Staubli VAL3: CopyFileContext.pgx

public program CopyFileContext(bool x_bRes (dimensions=1), string x_sFileSource (dimensions=1), string x_sFileDest (dimensions=1), num x_nStart (dimensions=1), num x_nEnd (dimensions=1))
  local num l_nIndex
  local num l_nNum
  local string l_sBuff
begin

  x_bRes=false
  if x_nEnd==-1
    x_nEnd=50000000
  endIf
  if x_sFileDest=="" or x_nStart<0 or x_nEnd<1 or x_nEnd<x_nStart or x_sFileDest==""
    return
  endIf
  if !$fileExists(x_sFileSource) or !$fileExists(x_sFileDest)
    return
  endIf


  nFileID=$fileOpen(x_sFileSource,"r")
  if nFileID<0 or nFileID>9
    return
  endIf

  nFile2ID=$fileOpen(x_sFileDest,"a")
  if nFile2ID<0 or nFile2ID>9
    return
  endIf


  l_nNum=1
  while true
    if $fileGet(nFileID,l_sBuff,l_nNum)!=1
      call CloseAllFile()
      return
    endIf
    if l_nIndex>=x_nStart and l_nIndex<=x_nEnd

      if $fileSet(nFile2ID,l_sBuff,l_nNum)!=1
        call CloseAllFile()
        return
      endIf
    endIf
    l_nIndex=l_nIndex+1
  endWhile

  call CloseAllFile()


end
